// TIA Portal V18 export
// export: Created 2025-12-01T17:51:09.9849749Z, ExportSetting None, DisplayName Totally Integrated Automation Portal, DisplayVersion V18 Update 5, DisplayName TIA Portal Openness, DisplayVersion V18 Update 5, DisplayName TIA Portal Teamcenter Gateway, DisplayVersion V18, DisplayName TIA Portal Version Control Interface, DisplayVersion V18, DisplayName STEP 7 Professional, DisplayVersion V18 Update 5, DisplayName STEP 7 Safety, DisplayVersion V18, DisplayName WinCC Professional, DisplayVersion V18 Update 5
DATA_BLOCK "Call_KeyenceCheckerIV_DB"   // DB2100
// stored: AutoNumber false, InstanceOfName Call_KeyenceCheckerIV, InstanceOfType FB
"Call_KeyenceCheckerIV"
   // VAR
   //    InsKeyenceCheckerIV3810A1 : "FB_KeyenceCheckerIV3";
   //    InsKeyenceCheckerIV3811A1 : "FB_KeyenceCheckerIV3";
   //    nIndex { S7_SetPoint := 'True'} : Int;
   // END_VAR
BEGIN
END_DATA_BLOCK
